% RSLogix 500 project Multiposition-Servo-Application.RSS, saved by version 8.40.00.08 %
PROJECT "UNTITLED"    % processor: Bul.1763 MicroLogix 1100 Series B %

PROGRAM FILES
  LAD 2   3 rungs
  LAD 3 "IO"  7 rungs
  LAD 4 "CONTROLS"  19 rungs

DATA FILES
  O0 OUTPUT  4 elements
  I1 INPUT  6 elements
  S2 STATUS  66 elements
  B3 BINARY  2 elements
  T4 TIMER  3 elements
  C5 COUNTER  1 elements
  R6 CONTROL  1 elements
  N7 INTEGER  3 elements
  F8 FLOAT  1 elements

LADDER 2
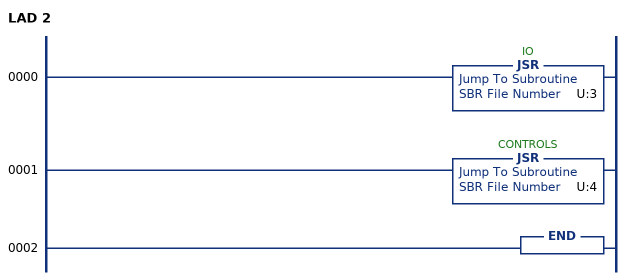
% Rung: 0 %
SOR JSR U:3 EOR
%   U:3  "IO" %
% Rung: 1 %
SOR JSR U:4 EOR
%   U:4  "CONTROLS" %
% Rung: 2 %
SOR END EOR

LADDER 3 "IO"
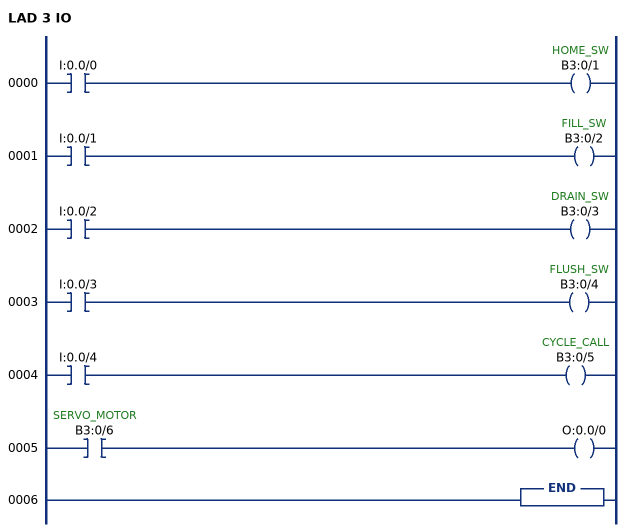
% Rung: 0 %
SOR XIC I:0.0/0 OTE B3:0/1 EOR
%   B3:0/1  HOME_SW %
% Rung: 1 %
SOR XIC I:0.0/1 OTE B3:0/2 EOR
%   B3:0/2  FILL_SW %
% Rung: 2 %
SOR XIC I:0.0/2 OTE B3:0/3 EOR
%   B3:0/3  DRAIN_SW %
% Rung: 3 %
SOR XIC I:0.0/3 OTE B3:0/4 EOR
%   B3:0/4  FLUSH_SW %
% Rung: 4 %
SOR XIC I:0.0/4 OTE B3:0/5 EOR
%   B3:0/5  CYCLE_CALL %
% Rung: 5 %
SOR XIC B3:0/6 OTE O:0.0/0 EOR
%   B3:0/6  SERVO_MOTOR %
% Rung: 6 %
SOR END EOR

LADDER 4 "CONTROLS"
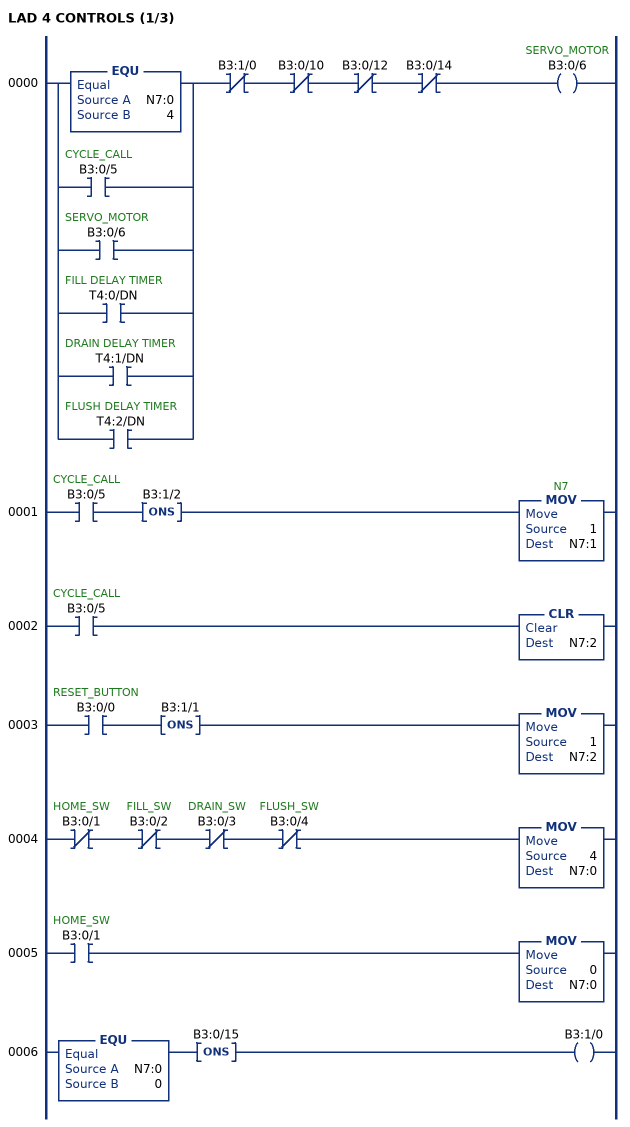
% Rung: 0 %
SOR BST EQU N7:0 4 NXB XIC B3:0/5 NXB XIC B3:0/6 NXB XIC T4:0/DN NXB XIC T4:1/DN NXB XIC T4:2/DN BND XIO B3:1/0 XIO B3:0/10 XIO B3:0/12 XIO B3:0/14 OTE B3:0/6 EOR
%   B3:0/5  CYCLE_CALL %
%   B3:0/6  SERVO_MOTOR %
%   T4:0  "FILL DELAY TIMER" %
%   T4:1  "DRAIN DELAY TIMER" %
%   T4:2  "FLUSH DELAY TIMER" %
% Rung: 1 %
SOR XIC B3:0/5 ONS B3:1/2 MOV 1 N7:1 EOR
%   B3:0/5  CYCLE_CALL %
%   N7:1  N7 %
% Rung: 2 %
SOR XIC B3:0/5 CLR N7:2 EOR
%   B3:0/5  CYCLE_CALL %
% Rung: 3 %
SOR XIC B3:0/0 ONS B3:1/1 MOV 1 N7:2 EOR
%   B3:0/0  RESET_BUTTON %
% Rung: 4 %
SOR XIO B3:0/1 XIO B3:0/2 XIO B3:0/3 XIO B3:0/4 MOV 4 N7:0 EOR
%   B3:0/1  HOME_SW %
%   B3:0/2  FILL_SW %
%   B3:0/3  DRAIN_SW %
%   B3:0/4  FLUSH_SW %
% Rung: 5 %
SOR XIC B3:0/1 MOV 0 N7:0 EOR
%   B3:0/1  HOME_SW %
% Rung: 6 %
SOR EQU N7:0 0 ONS B3:0/15 OTE B3:1/0 EOR

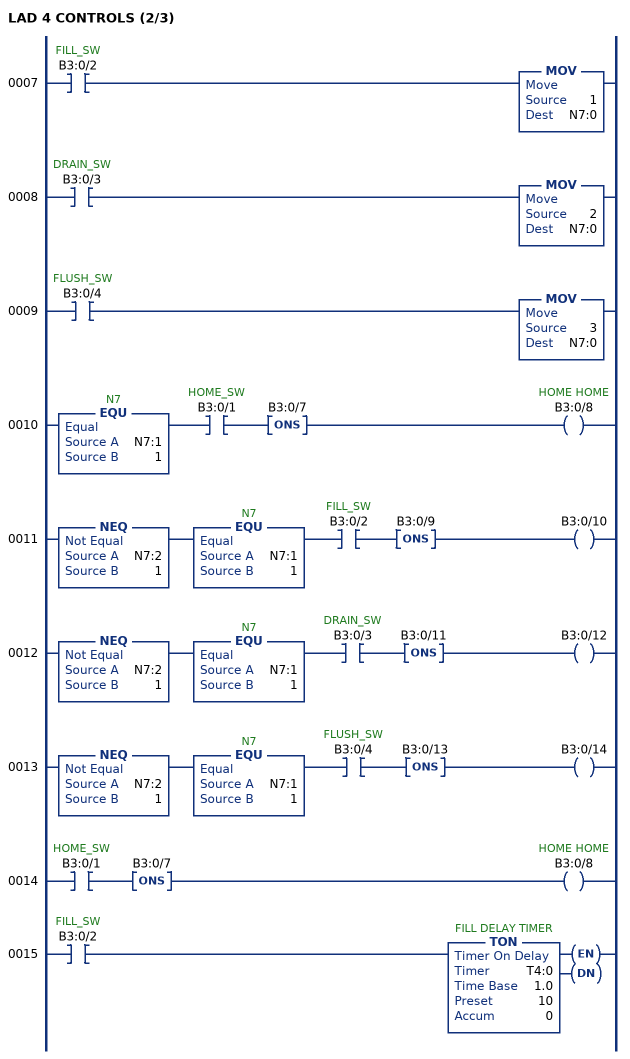
% Rung: 7 %
SOR XIC B3:0/2 MOV 1 N7:0 EOR
%   B3:0/2  FILL_SW %
% Rung: 8 %
SOR XIC B3:0/3 MOV 2 N7:0 EOR
%   B3:0/3  DRAIN_SW %
% Rung: 9 %
SOR XIC B3:0/4 MOV 3 N7:0 EOR
%   B3:0/4  FLUSH_SW %
% Rung: 10 %
SOR EQU N7:1 1 XIC B3:0/1 ONS B3:0/7 OTE B3:0/8 EOR
%   N7:1  N7 %
%   B3:0/1  HOME_SW %
%   B3:0/8  HOME  "HOME" %
% Rung: 11 %
SOR NEQ N7:2 1 EQU N7:1 1 XIC B3:0/2 ONS B3:0/9 OTE B3:0/10 EOR
%   N7:1  N7 %
%   B3:0/2  FILL_SW %
% Rung: 12 %
SOR NEQ N7:2 1 EQU N7:1 1 XIC B3:0/3 ONS B3:0/11 OTE B3:0/12 EOR
%   N7:1  N7 %
%   B3:0/3  DRAIN_SW %
% Rung: 13 %
SOR NEQ N7:2 1 EQU N7:1 1 XIC B3:0/4 ONS B3:0/13 OTE B3:0/14 EOR
%   N7:1  N7 %
%   B3:0/4  FLUSH_SW %
% Rung: 14 %
SOR XIC B3:0/1 ONS B3:0/7 OTE B3:0/8 EOR
%   B3:0/1  HOME_SW %
%   B3:0/8  HOME  "HOME" %
% Rung: 15 %
SOR XIC B3:0/2 TON T4:0 1.0 10 0 EOR
%   B3:0/2  FILL_SW %
%   T4:0  "FILL DELAY TIMER" %

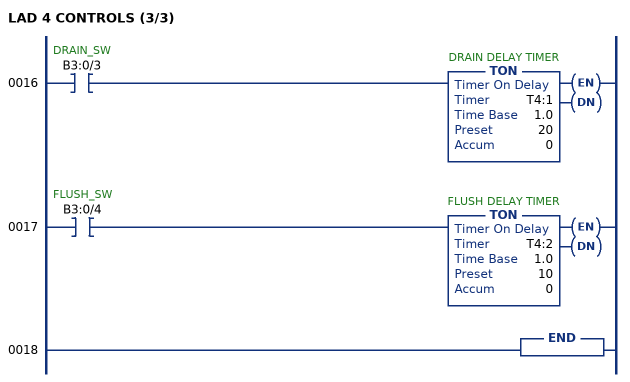
% Rung: 16 %
SOR XIC B3:0/3 TON T4:1 1.0 20 0 EOR
%   B3:0/3  DRAIN_SW %
%   T4:1  "DRAIN DELAY TIMER" %
% Rung: 17 %
SOR XIC B3:0/4 TON T4:2 1.0 10 0 EOR
%   B3:0/4  FLUSH_SW %
%   T4:2  "FLUSH DELAY TIMER" %
% Rung: 18 %
SOR END EOR

DATA TABLE (non-zero values as saved)
DATA T4
% .PRE .ACC %
% T4:0 % 10 0
% T4:1 % 20 0
% T4:2 % 10 0
